// TIA Portal V19 export
TYPE "Positioning_DOL_Machine_Manager"
// stored: Access Published
   STRUCT
      EnableStopDoorOpeningReq : Bool;
      EnableStopInPhase : Bool;
      EnableStopProgrammed : Bool;
      Control_ON : Bool;
      Minus : Bool;   // Move in negative direction
      Plus : Bool;   // Move in positive direction
      MoveToPos : Bool;   // Move to target position
      Pos : LReal;   // [mm] Target position
      Speed : LReal;   // [0-100] Target speed %
   END_STRUCT;
END_TYPE
